FUNCTION GetHypotenuse : LREAL
VAR_INPUT
	a : LREAL;
	b : LREAL;
END_VAR
VAR
	resultSquared : LREAL;
END_VAR

resultSquared := a * a + b * b;
GetHypotenuse := SQRT(resultSquared);

END_FUNCTION

(* stored: Version 1.1.0.1, ProductVersion 3.1.4024.12
   POU GetHypotenuse: Id {7f0d3285-114c-4b54-995b-47a8a1b05dc9}, SpecialFunc None *)
